FUNCTION F_Temperature : REAL
VAR_INPUT
	Input											: INT;
END_VAR
VAR
END_VAR

// Calvin - F_Temperature
// Rev 1.0 - March 3, 2023

F_Temperature										:= INT_TO_REAL(Input) / 10.0;

END_FUNCTION

(* stored: Version 1.1.0.1, ProductVersion 3.1.4024.11
   POU F_Temperature: Id {b0c73f2e-26d0-4c57-b376-becd046dc3ba}, SpecialFunc None *)
